// TIA Portal project "学习触点比较指令" (V15.1)

(* hardware
DEVICE "S7-1200 station_1"  S7-1200 Station
   slot 0: "Rack_0"  S7-1200 Rack  Rack  V1.0
   slot 1: "PLC_1"  CPU 1214C DC/DC/DC  6ES7 214-1AG40-0XB0  V4.2
*)

// ===== PLC "PLC_1"  CPU 1214C DC/DC/DC =====

VAR_GLOBAL   // PLC tag table "默认变量表"
   "Tag_1" AT %I0.0 : Bool;
   "Tag_2" AT %MD200 : Time;
   "Tag_3" AT %Q0.0 : Bool;
   "Tag_4" AT %MD204 : DInt;
   "Tag_5" AT %Q0.1 : Bool;
   "Tag_6" AT %M0.0 : Bool;
END_VAR

// folder: System blocks/Program resources

DATA_BLOCK "IEC_Timer_0_DB_3"   // DB5
{ S7_Optimized_Access := 'TRUE' }
AUTHOR : Simatic
FAMILY : IEC
NAME : IEC_TMR
VERSION : 1.0
// stored: InstanceOfName IEC_TIMER
"IEC_TIMER"
BEGIN
END_DATA_BLOCK

// folder: (top level)

ORGANIZATION_BLOCK "Main"   // OB1, LAD, ProgramCycle
TITLE = "Main Program Sweep (Cycle)"
{ S7_Optimized_Access := 'TRUE' }
VERSION : 0.1
   VAR_INPUT
      Initial_Call : Bool;   // Initial call of this OB
      Remanence : Bool;   // =True, if remanent data are available
   END_VAR
BEGIN

REGION Network 1: 利用定时器控制范围内的 输出 为1
   // 利用定时器的输出，给定时器一个常闭开关，可以做到复位的效果
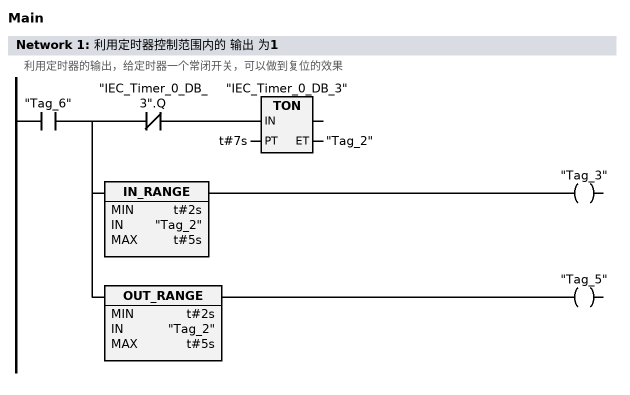
   "IEC_Timer_0_DB_3".TON(IN := "Tag_6" AND NOT "IEC_Timer_0_DB_3".Q, PT := t#7s, ET => "Tag_2");
   "Tag_3" := "Tag_6" AND (t#2s <= "Tag_2") AND ("Tag_2" <= t#5s);
   "Tag_5" := "Tag_6" AND (("Tag_2" < t#2s) OR ("Tag_2" > t#5s));
END_REGION
END_ORGANIZATION_BLOCK